Yaskawa INFORM job: BIGSLOW.JBI

/JOB
//NAME BIGSLOW
//POS
///NPOS 21,0,0,0,0,0
///TOOL 0
///POSTYPE PULSE
///PULSE
C00000=2276,25307,0,0,-64000,-407
C00001=1349,27065,0,0,-64000,-407
C00002=415,28819,0,0,-64000,-407
C00003=-504,30581,0,0,-64000,-407
C00004=-1447,32332,0,0,-64000,-407
C00005=-2358,34097,0,0,-64000,-407
C00006=-3308,35845,0,0,-64000,-407
C00007=-3626,37307,0,0,-64000,-407
C00008=-1627,37307,0,0,-64000,-407
C00009=373,37307,0,0,-64000,-407
C00010=2373,37307,0,0,-64000,-407
C00011=4373,37307,0,0,-64000,-407
C00012=6373,37307,0,0,-64000,-407
C00013=8374,37307,0,0,-64000,-407
C00014=7905,35781,0,0,-64000,-407
C00015=6964,34029,0,0,-64000,-407
C00016=6003,32286,0,0,-64000,-407
C00017=5103,30516,0,0,-64000,-407
C00018=4150,28770,0,0,-64000,-407
C00019=3223,27012,0,0,-64000,-407
C00020=2276,25307,0,0,-64000,-407
//INST
///DATE 2026/04/08 12:00
///ATTR SC,RW
///GROUP1 RB1
NOP
MOVJ C00000 VJ=2.00
MOVL C00001 V=20.0
MOVL C00002 V=20.0
MOVL C00003 V=20.0
MOVL C00004 V=20.0
MOVL C00005 V=20.0
MOVL C00006 V=20.0
MOVL C00007 V=20.0
MOVL C00008 V=20.0
MOVL C00009 V=20.0
MOVL C00010 V=20.0
MOVL C00011 V=20.0
MOVL C00012 V=20.0
MOVL C00013 V=20.0
MOVL C00014 V=20.0
MOVL C00015 V=20.0
MOVL C00016 V=20.0
MOVL C00017 V=20.0
MOVL C00018 V=20.0
MOVL C00019 V=20.0
MOVL C00020 V=20.0
END
